// TIA Portal V19 export
TYPE "LEXCHANGETRAY_typeNgConveyorEm_toHandlingXyzFeedback"
// stored: Access Published
   STRUCT
      transferEnable : Bool;   // 请求转移
      running : Bool;   // 运行中
   END_STRUCT;
END_TYPE
